{attribute 'qualified_only'}
VAR_GLOBAL
	TableRecord		: ARRAY [1..5,1..7] OF STRING;
	TODAY			: WORD;
	YESTERDAY		: WORD;
	LASTMONTH		: UINT;
	LASTYEAR		: UINT;
	
	DailyCnt_FG1	: INT;
	DailyCnt_FG2	: INT;
	DailyCnt_FG3	: INT;
	DailyCnt_FG4	: INT;
	MonthCnt		: UINT;
	YearCnt			: UINT;
END_VAR

(* stored: Version 1.1.0.1, ProductVersion 3.1.4024.12
   GVL GVL: Id {91cce4c8-d258-4ec1-a4bf-b4e621e39a91} *)
